// Minimal concrete probe for the base classes (Fraktal_QuickStart_and_Suite.md §1).
// Its ONLY logic is _M_Dispatch — everything else is inherited, which is the point.
FUNCTION_BLOCK FB_ProbeCM EXTENDS FB_ControlModuleBase
VAR_INPUT
    SimDone  : BOOL;
    SimFault : BOOL;
END_VAR

Cyclic();

METHOD Setup : BOOL
VAR_INPUT
    Name : STRING(80);
END_VAR
_M_SetName(Name);
Setup := TRUE;
END_METHOD

METHOD PROTECTED _M_Dispatch
_M_TagCommand(Id := 1, Label := 'PROBE');   // §8.11.4(a) — the one-line command tag
IF SimFault THEN
    _M_Fault(E_Reason.TEST_FAULT, 'probe fault');
ELSIF SimDone THEN
    _M_Complete();
END_IF
END_METHOD

END_FUNCTION_BLOCK

(* stored: Version 1.1.0.1, ProductVersion 3.1.4024.12
   POU FB_ProbeCM: Id {ace2ffef-da6f-4500-bb16-d6b5e668246d}, SpecialFunc None
   Method Setup: Id {fa777fc7-9e8d-4c24-aab9-7b0fc5bce9d1}
   Method _M_Dispatch: Id {09dda4aa-ea32-4a00-b61d-5b786f9f2569} *)
